// TIA Portal project "S7-400" (V15)

(* hardware
DEVICE "S7-400 station_1"  S7-400 station
   slot 0: "UR1_0"  UR1  6ES7 400-1TA01-0AA0
   slot 1: "PS 407 4A_1"  PS 407 4A  6ES7 407-0DA02-0AA0
   slot 1: "DP interface_1"  X2  6ES7 964-2AA04-0AB0
   slot 2: "PLC_1"  CPU 414-3 PN/DP  6ES7 414-3EM05-0AB0  V5.3
      slot 2: "MPI/DP interface_1"  X1
      slot 5: "PROFINET interface_1"  PN-IO
         slot 1: "Port_1"  Port
         slot 2: "Port_2"  Port
   slot 4: "DI 16x24VDC_1"  DI16 x 24VDC interrupt  6ES7 421-7BH01-0AB0
   slot 5: "DO 16x24VDC/2A_1"  DO16 x 24VDC / 2A  6ES7 422-1BH11-0AA0
   slot 9: "CP 443-5 Ext_1"  CP 443-5 Extended  6GK7 443-5DX05-0XE0  V7.0
   slot 10: "CP 443-5 Ext_2"  CP 443-5 Extended  6GK7 443-5DX05-0XE0  V7.0
   slot 11: "CP 443-5 Ext_3"  CP 443-5 Extended  6GK7 443-5DX05-0XE0  V7.0
DEVICE "ET 200S station_1"  ET 200S station
   slot 0: "Rack_0"  Rail
   slot 2: "DP interface_1"  DP  6ES7 138-4HA00-0AB0  V1.0
   slot 2: "PLC_2"  IM151-7 F-CPU  6ES7 151-7FA20-0AB0  V2.6
      slot 1: "MPI/DP interface_1"  X1
   slot 4: "PM-E 24VDC_1"  PM-E 24VDC  6ES7 138-4CA01-0AA0
   slot 5: "2DI x 24VDC ST_1"  2DI x 24VDC ST  6ES7 131-4BB01-0AA0
*)

// ===== PLC "PLC_1"  CPU 414-3 PN/DP =====

VAR_GLOBAL   // PLC tag table "Default tag table"
   "OUT_1" AT %M100.0 : Bool;
   "START" AT %M10.1 : Bool;
   "STOP" AT %M10.2 : Bool;
   "START_2" AT %M10.3 : Bool;
   "STOP_2" AT %M10.4 : Bool;
   "OUT_2" AT %M100.1 : Bool;
   "START_03" AT %M10.5 : Bool;
   "STOP_03" AT %M10.6 : Bool;
   "OUT_3" AT %M100.2 : Bool;
   "SS_TRIG_3" AT %M10.7 : Bool;
   "TIMER_FB2" AT %T1 : Timer;
END_VAR

VAR_GLOBAL   // PLC tag table "Tag table_1"
   "FB_1.DB2.IN_1" AT %M101.0 : Bool;
   "FB_1.DB2.IN_2" AT %M101.1 : Bool;
   "FB_1.DB2.IN_3" AT %M101.2 : Bool;
   "FB_1.DB2.IN_4" AT %M101.3 : Bool;
   "FB_1.DB2.IN_5" AT %M101.4 : Bool;
   "FB_1.DB2.IN_6" AT %M101.5 : Bool;
   "FB_1.DB2.OUT" AT %M201.6 : Bool;
   "FB_2.DB3.OUT" AT %M201.7 : Bool;
   "FB_2.DB3.ENA" AT %M101.6 : Bool;
   "FB_2.DB3.RST" AT %M101.7 : Bool;
   "FB_2.DB3.CR_VAL_BI" AT %ID202 : Time;
END_VAR

DATA_BLOCK "BD1"   // DB1
{ S7_Optimized_Access := 'FALSE' }
VERSION : 0.1
BEGIN
END_DATA_BLOCK

DATA_BLOCK "STL_FB_DB"   // DB2
{ S7_Optimized_Access := 'FALSE' }
VERSION : 0.1
// stored: InstanceOfName STL_FB
"STL_FB"
BEGIN
END_DATA_BLOCK

DATA_BLOCK "STL_FB_TIMER_DB"   // DB3
{ S7_Optimized_Access := 'FALSE' }
VERSION : 0.1
// stored: InstanceOfName STL_FB_TIMER
"STL_FB_TIMER"
BEGIN
END_DATA_BLOCK

DATA_BLOCK "STL_FB_TIMER_DB_1"   // DB4
{ S7_Optimized_Access := 'FALSE' }
VERSION : 0.1
// stored: InstanceOfName STL_FB_TIMER
"STL_FB_TIMER"
BEGIN
END_DATA_BLOCK

DATA_BLOCK "STL_FB_TIMER_DB_2"   // DB5
{ S7_Optimized_Access := 'FALSE' }
VERSION : 0.1
// stored: InstanceOfName STL_FB_TIMER
"STL_FB_TIMER"
BEGIN
END_DATA_BLOCK

FUNCTION_BLOCK "STL_FB"   // FB1, STL
{ S7_Optimized_Access := 'FALSE' }
VERSION : 0.1
   VAR_INPUT
      IN_1 : Bool;
      IN_2 : Bool;
      IN_3 : Bool;
      IN_4 : Bool;
      IN_5 : Bool;
      IN_6 : Bool;
   END_VAR
   VAR_OUTPUT
      OUT : Bool;
   END_VAR
BEGIN

REGION Network 1
         A     #IN_1;
         A     #IN_2;
         O;
         A     #IN_3;
         A     #IN_4;
         O     #IN_5;
         AN    #IN_6;
         =     #OUT;
END_REGION
END_FUNCTION_BLOCK

FUNCTION_BLOCK "STL_FB_TIMER"   // FB2, STL
{ S7_Optimized_Access := 'FALSE' }
VERSION : 0.1
   VAR_INPUT
      ENA_FC_TIMER : Bool;
      RESER_TIMER : Bool;
      TV_TIMER : Time;
   END_VAR
   VAR_OUTPUT
      OUT : Bool;
      CR_VAL_TIMER : Time;
   END_VAR
   VAR_TEMP
      SIMPLE_TIMER : Time;
   END_VAR
   VAR CONSTANT
      "TIMER" : Time;
   END_VAR
BEGIN

REGION Network 1
   // SIMPLE BLOCK STTL TIMER
         FR    "TIMER_FB2";
         A     #ENA_FC_TIMER;  // ENABLE TIMER SIMPLE FUN TION BLOCK
         L     #TV_TIMER;  // SET 10S PRESET TIME IN ACU
         SD    "TIMER_FB2";  // START ON DELAY TIMER_FB
         A     #RESER_TIMER;
         R     "TIMER_FB2";  // RESET TIMER TIMER_FB
         A     "TIMER_FB2";
         =     #OUT;
         L     "TIMER_FB2";
         T     #CR_VAL_TIMER;  // CURRENT VALUE FOR TIMER_FB2
END_REGION
END_FUNCTION_BLOCK

FUNCTION "FUN_2599" : Void   // FC1, STL
{ S7_Optimized_Access := 'FALSE' }
VERSION : 0.1
BEGIN
END_FUNCTION

ORGANIZATION_BLOCK "Main"   // OB1, LAD
TITLE = "Main Program Sweep (Cycle)"
{ S7_Optimized_Access := 'FALSE' }
VERSION : 0.1
   VAR_TEMP
      OB1_EV_CLASS : Byte;   // Bits 0-3 = 1 (Coming event), Bits 4-7 = 1 (Event class 1)
      OB1_SCAN_1 : Byte;   // 1 (Cold restart scan 1 of OB 1), 3 (Scan 2-n of OB 1)
      OB1_PRIORITY : Byte;   // Priority of OB Execution
      OB1_OB_NUMBR : Byte;   // 1 (Organization block 1, OB1)
      OB1_RESERVED_1 : Byte;   // Reserved for system
      OB1_RESERVED_2 : Byte;   // Reserved for system
      OB1_PREV_CYCLE : Int;   // Cycle time of previous OB1 scan (milliseconds)
      OB1_MIN_CYCLE : Int;   // Minimum cycle time of OB1 (milliseconds)
      OB1_MAX_CYCLE : Int;   // Maximum cycle time of OB1 (milliseconds)
      OB1_DATE_TIME : Date_And_Time;   // Date and time OB1 started
   END_VAR
BEGIN

REGION Network 1 (STL)
         A     "START";
         AN    "STOP";
         =     "OUT_1";
END_REGION

REGION Network 2 (STL)
   // NHAN TU TRANG THAI RELAY
         O     "START_2";
         O     "OUT_2";
         AN    "STOP_2";
         =     "OUT_2";
END_REGION

REGION Network 3 (STL)
   // LENH A() KET NOI CAC TRANG THAI AND TICH HOP LAI VOI NHAU
         A(;
         O     "START_03";
         O     "OUT_3";
         );
         A(;
         ON    "STOP_03";
         O     "SS_TRIG_3";
         );
         =     "OUT_3";
END_REGION

REGION Network 4
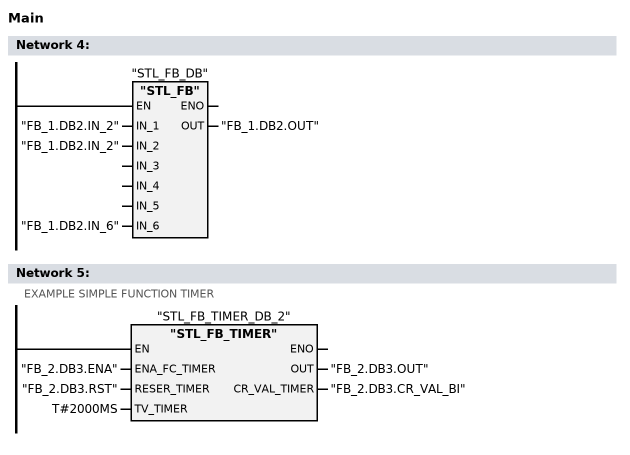
   RUNG wire#powerrail
      "STL_FB_DB"(IN_1 := "FB_1.DB2.IN_2", IN_2 := "FB_1.DB2.IN_2", IN_3 :=, IN_4 :=, IN_5 :=, IN_6 := "FB_1.DB2.IN_6", OUT => "FB_1.DB2.OUT")
   END_RUNG
   // the same network as SCL:
   "STL_FB_DB"(IN_1 := "FB_1.DB2.IN_2", IN_2 := "FB_1.DB2.IN_2", IN_6 := "FB_1.DB2.IN_6", OUT => "FB_1.DB2.OUT");   // "STL_FB"
END_REGION

REGION Network 5
   // EXAMPLE SIMPLE FUNCTION TIMER
   RUNG wire#powerrail
      "STL_FB_TIMER_DB_2"(ENA_FC_TIMER := "FB_2.DB3.ENA", RESER_TIMER := "FB_2.DB3.RST", TV_TIMER := T#2000MS, OUT => "FB_2.DB3.OUT", CR_VAL_TIMER => "FB_2.DB3.CR_VAL_BI")
   END_RUNG
   // the same network as SCL:
   "STL_FB_TIMER_DB_2"(ENA_FC_TIMER := "FB_2.DB3.ENA",   // "STL_FB_TIMER"
                       RESER_TIMER := "FB_2.DB3.RST",
                       TV_TIMER := T#2000MS,
                       OUT => "FB_2.DB3.OUT",
                       CR_VAL_TIMER => "FB_2.DB3.CR_VAL_BI");
END_REGION
END_ORGANIZATION_BLOCK

// ===== PLC "PLC_2"  IM151-7 F-CPU =====

ORGANIZATION_BLOCK "Main"   // OB1, LAD
TITLE = "Main Program Sweep (Cycle)"
{ S7_Optimized_Access := 'FALSE' }
VERSION : 0.1
   VAR_TEMP
      OB1_EV_CLASS : Byte;   // Bits 0-3 = 1 (Coming event), Bits 4-7 = 1 (Event class 1)
      OB1_SCAN_1 : Byte;   // 1 (Cold restart scan 1 of OB 1), 3 (Scan 2-n of OB 1)
      OB1_PRIORITY : Byte;   // Priority of OB Execution
      OB1_OB_NUMBR : Byte;   // 1 (Organization block 1, OB1)
      OB1_RESERVED_1 : Byte;   // Reserved for system
      OB1_RESERVED_2 : Byte;   // Reserved for system
      OB1_PREV_CYCLE : Int;   // Cycle time of previous OB1 scan (milliseconds)
      OB1_MIN_CYCLE : Int;   // Minimum cycle time of OB1 (milliseconds)
      OB1_MAX_CYCLE : Int;   // Maximum cycle time of OB1 (milliseconds)
      OB1_DATE_TIME : Date_And_Time;   // Date and time OB1 started
   END_VAR
BEGIN
END_ORGANIZATION_BLOCK